% RSLogix 500 project task5.RSS, saved by version 8.30.00.16 %
PROJECT "UNTITLED"    % processor: Bul.1763 MicroLogix 1100 Series B %

PROGRAM FILES
  LAD 2   7 rungs

DATA FILES
  O0 OUTPUT  4 elements
  I1 INPUT  6 elements
  S2 STATUS  66 elements
  B3 BINARY  1 elements
  T4 TIMER  1 elements
  C5 COUNTER  1 elements
  R6 CONTROL  1 elements
  N7 INTEGER  1 elements
  F8 FLOAT  1 elements

LADDER 2
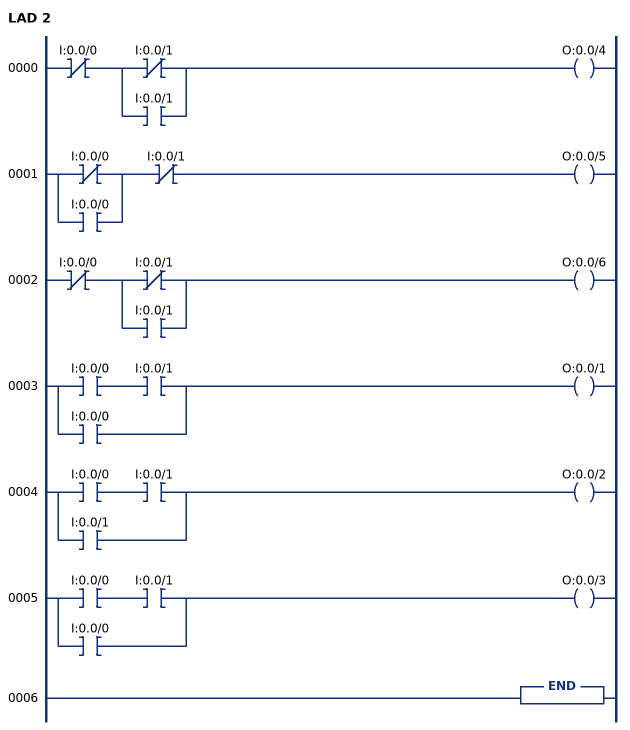
% Rung: 0 %
SOR XIO I:0.0/0 BST XIO I:0.0/1 NXB XIC I:0.0/1 BND OTE O:0.0/4 EOR
% Rung: 1 %
SOR BST XIO I:0.0/0 NXB XIC I:0.0/0 BND XIO I:0.0/1 OTE O:0.0/5 EOR
% Rung: 2 %
SOR XIO I:0.0/0 BST XIO I:0.0/1 NXB XIC I:0.0/1 BND OTE O:0.0/6 EOR
% Rung: 3 %
SOR BST XIC I:0.0/0 XIC I:0.0/1 NXB XIC I:0.0/0 BND OTE O:0.0/1 EOR
% Rung: 4 %
SOR BST XIC I:0.0/0 XIC I:0.0/1 NXB XIC I:0.0/1 BND OTE O:0.0/2 EOR
% Rung: 5 %
SOR BST XIC I:0.0/0 XIC I:0.0/1 NXB XIC I:0.0/0 BND OTE O:0.0/3 EOR
% Rung: 6 %
SOR END EOR
